FUNCTION_BLOCK PID (* Composite Function Block Type *)
  (* Standard: 61499-2 *)
  (* Version 0.0, 1/20/2026, Schneider Electric, template *)
  PACKAGE Hidryco.HidrycoLib;
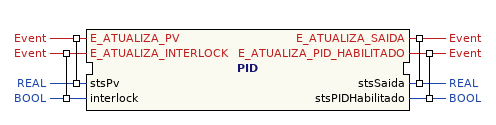
  EVENT_INPUT
    E_ATUALIZA_PV WITH stsPv;
    E_ATUALIZA_INTERLOCK WITH interlock;
  END_EVENT
  EVENT_OUTPUT
    E_ATUALIZA_SAIDA WITH stsSaida;
    E_ATUALIZA_PID_HABILITADO WITH stsPIDHabilitado;
  END_EVENT
  VAR_INPUT
    stsPv : REAL;
    interlock : BOOL;
  END_VAR
  VAR_OUTPUT
    stsSaida : REAL;
    stsPIDHabilitado : BOOL;
  END_VAR
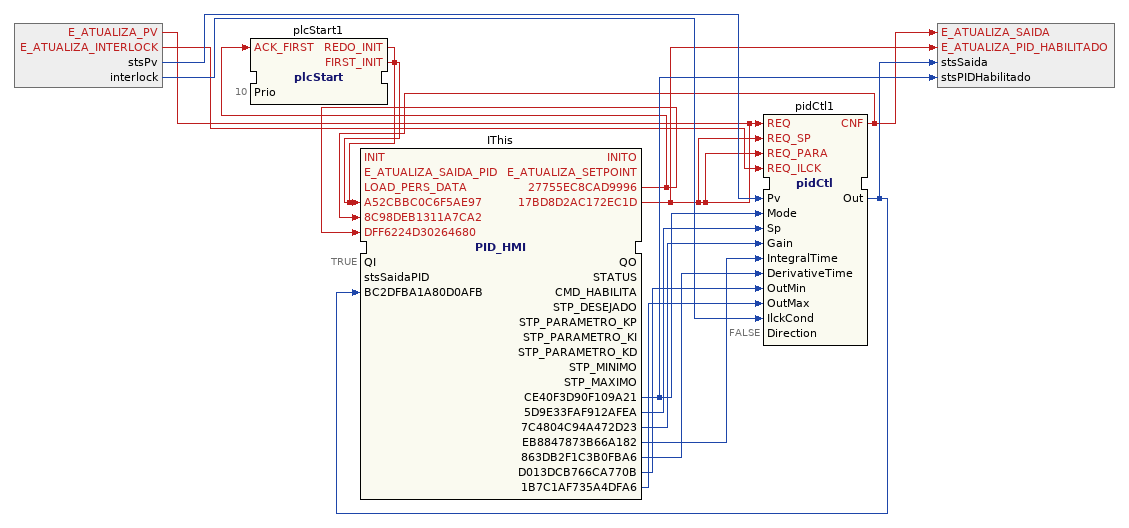
  FBS
    pidCtl1 : pidCtl(Direction := FALSE);
    IThis : PID_HMI(QI := TRUE);
    plcStart1 : plcStart(Prio := 10);
  END_FBS
  EVENT_CONNECTIONS
    E_ATUALIZA_PV TO pidCtl1.REQ;
    plcStart1.REDO_INIT TO IThis.A52CBBC0C6F5AE97;
    plcStart1.FIRST_INIT TO IThis.A52CBBC0C6F5AE97;
    pidCtl1.CNF TO IThis.8C98DEB1311A7CA2;
    IThis.27755EC8CAD9996 TO IThis.DFF6224D30264680;
    IThis.17BD8D2AC172EC1D TO pidCtl1.REQ;
    IThis.17BD8D2AC172EC1D TO pidCtl1.REQ_SP;
    IThis.17BD8D2AC172EC1D TO pidCtl1.REQ_PARA;
    IThis.27755EC8CAD9996 TO plcStart1.ACK_FIRST;
    pidCtl1.CNF TO E_ATUALIZA_SAIDA;
    IThis.17BD8D2AC172EC1D TO E_ATUALIZA_PID_HABILITADO;
    E_ATUALIZA_INTERLOCK TO pidCtl1.REQ_ILCK;
  END_CONNECTIONS
  DATA_CONNECTIONS
    stsPv TO pidCtl1.Pv;
    pidCtl1.Out TO IThis.BC2DFBA1A80D0AFB;
    IThis.CE40F3D90F109A21 TO pidCtl1.Mode;
    IThis.5D9E33FAF912AFEA TO pidCtl1.Sp;
    IThis.7C4804C94A472D23 TO pidCtl1.Gain;
    IThis.EB8847873B66A182 TO pidCtl1.IntegralTime;
    IThis.863DB2F1C3B0FBA6 TO pidCtl1.DerivativeTime;
    IThis.D013DCB766CA770B TO pidCtl1.OutMin;
    IThis.1B7C1AF735A4DFA6 TO pidCtl1.OutMax;
    pidCtl1.Out TO stsSaida;
    IThis.CE40F3D90F109A21 TO stsPIDHabilitado;
    interlock TO pidCtl1.IlckCond;
  END_CONNECTIONS
END_FUNCTION_BLOCK
